// TIA Portal V20 export
VAR_GLOBAL   // PLC tag table "Analog_Inputs"
   AI_LaserPowerMeter AT %IW412 : Word;
   AI_AxisB_ClampingPart AT %IW414 : Word;
   AI_LaserAirPressureProcess AT %IW416 : Word;
   AI_InletAirPressure AT %IW418 : Word;
   AI_AmbiantTemperature AT %IW428 : Word;
   AI_MachineTemperature AT %IW430 : Word;
   AI_ColdWaterTemperatureInput AT %IW432 : Word;
   AI_ColdWaterTemperatureOutput AT %IW434 : Word;
   AI_X_AxisTemperaturePT1000 AT %IW436 : Word;
   AI_Y_AxisTemperaturePT1000 AT %IW438 : Word;
   "AI_X_ AxisTemperaturePTC" AT %IW440 : Word;
   "AI_Y_ AxisTemperaturePTC" AT %IW442 : Word;
   AI_NozzleOverpressure AT %IW444 : Word;
   AI_OpticalPathOverpressure AT %IW446 : Word;
   AI_LaserHeadOverpressure AT %IW448 : Word;
   AI_ZL_AxisOverpressure AT %IW450 : Word;
   AI_XY_AxisOverpressure AT %IW452 : Word;
   AI_LeftAspiration AT %IW454 : Word;
   AI_RightAspiration AT %IW456 : Word;
   AI_FreeIW458 AT %IW458 : Word;
   AI_ClimTemperature AT %IW480 : Word;
   AI_FreeIW482 AT %IW482 : Word;
   AI_FreeIW484 AT %IW484 : Word;
   AI_FreeIW486 AT %IW486 : Word;
   AI_SensorControllerStation1 AT %IW460 : Word;
   AI_CabinetTemperature AT %IW462 : Word;
   AI_FreeIW464 AT %IW464 : Word;
   AI_FreeIW466 AT %IW466 : Word;
END_VAR
